(* IEC 61131-3 sources: teller/JD_Teller_LC2_V11/Class/SV_Help, 1 file *)

(* ---- SV_Help.st ---- *)
(*!
<Class
	Name               = "SV_Help"
	Revision           = "0.0"
	RealtimeTask       = "false"
	CyclicTask         = "false"
	DefCyclictime      = "50 ms"
	BackgroundTask     = "false"
	DefBackgroundIndex = "2147483392"
	Sigmatek           = "false"
	OSInterface        = "false"
	HighPriority       = "false"
	Automatic          = "false"
	UpdateMode         = "Prescan"
	SharedCommandTable = "true"
	Objectsize         = "(450,480)">
	<Channels>
		<Server Name="ClassSvr" Visualized="true" Initialize="false" WriteProtected="true" Retentive="false"/>
		<Server Name="Help_Conveyor_LSU_Svr" Visualized="true" Initialize="false" WriteProtected="false" Retentive="false"/>
		<Server Name="Help_Doos_Opslag_Svr" Visualized="true" Initialize="false" WriteProtected="false" Retentive="false"/>
		<Server Name="Help_Kicker_Sprayer_Uitrichter_Svr" Visualized="true" Initialize="false" WriteProtected="false" Retentive="false"/>
		<Server Name="Help_Main_Aantal_Dozen_Svr" Visualized="true" Initialize="false" WriteProtected="false" Retentive="false"/>
		<Server Name="Help_Main_Buttons" Visualized="true" Initialize="false" WriteProtected="false" Retentive="false"/>
		<Server Name="Help_TeachIn_Svr" Visualized="true" Initialize="false" WriteProtected="false" Retentive="false"/>
	</Channels>
</Class>
*)
SV_Help : CLASS
  //Servers:
	ClassSvr 	: SvrChCmd_DINT;
	Help_Doos_Opslag_Svr 	: SvrCh_DINT;
	Help_Main_Aantal_Dozen_Svr 	: SvrCh_DINT;
	Help_Kicker_Sprayer_Uitrichter_Svr 	: SvrCh_DINT;
	Help_Conveyor_LSU_Svr 	: SvrCh_DINT;
	Help_TeachIn_Svr 	: SvrCh_DINT;
	Help_Main_Buttons 	: SvrCh_DINT;
  //Clients:
  //Variables:
  //Functions:
  //Tables:
	FUNCTION @STD
		VAR_OUTPUT
			ret_code	: CONFSTATES;
		END_VAR;
	FUNCTION GLOBAL TAB @CT_;
END_CLASS;
